Staubli VAL3: onF1Event.pgx

program onF1Event()
  local bool l_NoBox
  local bool l_bStop
  local string l_sDynamicStu[3]
  local num l_n
  local string l_sMessage
begin
  // look if the bButton is enable
  if bButton[0]
    if cycleStatus:bIsHome
       call language2:message(l_sMessage,58)
       popUpMsg(l_sMessage)
      return
    endIf
    call set:_IsUseingBox(l_NoBox)
    if l_NoBox==true
           call language2:message(l_sMessage,59)
       popUpMsg(l_sMessage)
      return
    endIf
    if workingMode( )==1 and !cycleStatus:bCycle  and !cycleStatus:bIsHome and !l_NoBox
      //      call use:timerDialog("请选择夹爪号,默认为1",2)
      //      call _setToolType()
      taskCreate "GOHOME",100,set:GOHOME()
      wait(taskStatus("GOHOME")==1)
      cls()

      cycleStatus:bHoming=true
      l_sDynamicStu[0]=">"
      l_sDynamicStu[1]=">>"
      l_sDynamicStu[2]=">>>"
      set:sHomingStatus=""
      do
        // set the menu
        //call use:setMenu(sMenu,true,-1)
        call use:type(32,13,"STOP ")
        nKey=getKey()
        // REFRESH
        if nKey==277
          stopMove()
          taskKill("GOHOME")
          wait(taskStatus("GOHOME")==-1)
          resetMotion( )
          l_bStop=true
        endIf
          call language2:message(l_sMessage,60)
        call use:timerDialog(l_sMessage+l_sDynamicStu[l_n]+"#"+set:sHomingStatus,0.5)
        if l_n==2
          l_n=0
        else
          l_n=l_n+1
        endIf
        delay(0.3)
      until l_bStop or  cycleStatus:bHoming==false  or cycleStatus:bIsHome
      cycleStatus:bHoming=false
      use:bUseRefresh =true
      cls()
    endIf
  endIf
end
